INTERFACE I_DigitalInput

PROPERTY PUBLIC State : BOOL
GET
END_GET
END_PROPERTY

END_INTERFACE

(* stored: Version 1.1.0.1, ProductVersion 3.1.4024.5
   Itf I_DigitalInput: Id {c82f3116-0b65-49b8-935b-f6052aa7425a}
   Property State: Id {7300b579-0868-4226-a0b7-1fba4de47ec4}
   Get Get: Id {b294ea88-a0d7-45b2-bdab-55810acf1b37} *)
